(* CODESYS project Industy_RECOVERED_2026-05-19T08-51-21.project

Project tree, tasks and I/O mapping:
  Device : CODESYS Control Win V3 x64, CODESYS, version 3.5.22.10
    application Application
      libraries: Standard, 3.5.22.0 (System)
      task MainTask (cyclic, interval t#20ms, priority 1) calls PLC_PRG
      DUTs (Data Types)/
        data type ST_AreaStatus
      program PLC_PRG [ST]
      Processes/
        program POU_07_Packaging [ST]
        program POU_03_Dryer [ST]
        program POU_04_Shelling [ST]
        program POU_01_Receiving [ST]
        program POU_02_Husking [ST]
        program POU_06_Treating [ST]
        program POU_05_Conditioning [ST]
      Blocks/
        function block POU_Vibration_Sensor [ST]
        function block POU_Flow_Sensor [ST]
        function block POU_Motor [ST]
      Symbols
*)

// Device/Application/DUTs (Data Types)/ST_AreaStatus
TYPE ST_AreaStatus :
STRUCT
	Running : BOOL;
	Stopped : BOOL;
	Failure : BOOL;
	Counters : DINT;
END_STRUCT
END_TYPE

// Device/Application/PLC_PRG
PROGRAM PLC_PRG
VAR

END_VAR

POU_01_Receiving();
POU_02_Husking();
POU_03_Dryer();
POU_04_Shelling();
POU_05_Conditioning();
POU_06_Treating();
POU_07_Packaging();

END_PROGRAM

// Device/Application/Processes/POU_01_Receiving
PROGRAM POU_01_Receiving
VAR
	CNV_001 : POU_Motor();
	
	Process_State : DINT;
	H_Start_Process : BOOL;
	
	Weight_Load : REAL;
	Truck_Counter : DINT;
	
	Timer_Truck_Discharge : TON;
	
END_VAR

CNV_001();

CASE Process_State OF
	0: //Initial State - Stopped
		CNV_001.I_Auto_Start := FALSE;
		IF H_Start_Process THEN
			Process_State := 1;
		END_IF
		H_Start_Process := FALSE;
	
	1: //Weighting Truck
		IF Truck_Counter MOD 2 = 0 THEN
			Weight_Load := Weight_Load + 2568;
		ELSE
			Weight_Load := Weight_Load - 1432;
		END_IF
		Truck_Counter := Truck_Counter + 1;
		Process_State := 2;
		
	2: //Start Unloading Truck
		Timer_Truck_Discharge(IN := TRUE, PT := T#2M);
		CNV_001.I_Auto_Start := TRUE;
		IF Timer_Truck_Discharge.Q THEN //When Finished receiving
			CNV_001.I_Auto_Start := FALSE;
			Timer_Truck_Discharge.IN := FALSE;
			Process_State := 0;
		END_IF		
		
	ELSE //Error
		Process_State := -1;
END_CASE

END_PROGRAM

// Device/Application/Blocks/POU_Motor
FUNCTION_BLOCK PUBLIC POU_Motor
VAR_INPUT
	I_Auto_Start : BOOL;
END_VAR
VAR_OUTPUT
	O_Start_Motor : BOOL;
END_VAR
VAR
	
END_VAR

IF I_Auto_Start THEN
	O_Start_Motor := TRUE;
ELSE
	O_Start_Motor := FALSE;
END_IF

END_FUNCTION_BLOCK

// Device/Application/Processes/POU_02_Husking
PROGRAM POU_02_Husking

VAR
	Process_Status : DINT;
	Receiving_Status : DINT;
	CNV_002 : POU_Motor;
	HUS_001 : POU_Motor;
	Bins_Counter : DINT;
	
	Timer_End_of_Line : TON;

END_VAR

Receiving_Status := POU_01_Receiving.Process_State;

CASE Process_Status OF
	0: //Initial State - Stopped
		HUS_001.I_Auto_Start := FALSE;
		CNV_002.I_Auto_Start := FALSE;
		IF Receiving_Status = 1 THEN
			Process_Status := 1;
		END_IF

	1: //Starting Motors to husk 
		HUS_001.I_Auto_Start := TRUE;
		CNV_002.I_Auto_Start := TRUE;
		IF Receiving_Status = 2 THEN
			Process_Status := 2;
		END_IF
		
	2: //Husking Corn
		IF POU_01_Receiving.Timer_Truck_Discharge.Q THEN
			Timer_End_of_Line(IN := TRUE, PT := T#1M);
			IF Timer_End_of_Line.Q THEN
				HUS_001.I_Auto_Start := FALSE;
				CNV_002.I_Auto_Start := FALSE;
				Process_Status := 3;
			END_IF
		END_IF
		
	3: //Bin Dryer Full
		Bins_Counter := Bins_Counter + 1;
		Timer_End_of_Line.IN := FALSE;
		Process_Status := 0;
		
	ELSE //Error
		Process_Status := -1;		
END_CASE

END_PROGRAM

// Device/Application/Processes/POU_03_Dryer
PROGRAM POU_03_Dryer
VAR
	Husking_Status : DINT;
	Process_Status : DINT;
	Dryed_Bins : DINT;
	
	BLR_001 : POU_Motor;
	CNV_003 : POU_Motor;
	
	Air_Temp : REAL;
	Grain_Humidity : REAL;	
	
	Timer_End_of_Line : TON;
	Timer_Humi_Decreaser : TP;
	
	
END_VAR

Husking_Status := POU_02_Husking.Process_Status;

CASE Process_Status OF
	0: //Initial_Case - Stopped
		BLR_001.I_Auto_Start := FALSE;
		CNV_003.I_Auto_Start := FALSE;
		IF Husking_Status = 3 THEN
			Process_Status := 1;
		END_IF
		
	1: //Starting Dryer
		BLR_001.I_Auto_Start := TRUE;
		Grain_Humidity := 35.0;
		Air_Temp := 45.0;
		Process_Status := 2;
	2: //Drying Corn
		Timer_Humi_Decreaser(IN := NOT Timer_Humi_Decreaser.Q, PT := T#1M);
		WHILE Process_Status = 2 DO
			IF Grain_Humidity <= 13.0 AND Air_Temp = 45 THEN
				Process_Status := 3;
			ELSE
				IF Timer_Humi_Decreaser.Q THEN
					Grain_Humidity := Grain_Humidity - 0.35;					
				END_IF
			END_IF						
		END_WHILE
	
	3: // Corn Dry
		BLR_001.I_Auto_Start := FALSE;
		CNV_003.I_Auto_Start := TRUE;
		Timer_End_of_Line(IN := TRUE, PT := T#1M);
		IF Timer_End_of_Line.Q THEN
			CNV_003.I_Auto_Start := FALSE;
			Process_Status := 4;
		END_IF
		
	4: //Bin Empty
		Dryed_Bins := Dryed_Bins + 1;
		Timer_End_of_Line.IN := FALSE;
		Process_Status := 0;
		
	ELSE //Error
		Process_Status := -1;
END_CASE

END_PROGRAM

// Device/Application/Processes/POU_04_Shelling
PROGRAM POU_04_Shelling
VAR
	Dryer_Status : DINT;
	Process_Status : DINT;
	
	Sheller_RPM : REAL;
	Grain_Flow : REAL;
	
	SHL_001 : POU_Motor;
	CNV_004 : POU_Motor;
	
	Timer_Acc_Sheller : TP;
	Timer_End_of_Line : TON;
	
	Flow_Sensor : POU_Flow_Sensor;
	
END_VAR

Dryer_Status := POU_03_Dryer.Process_Status;
Flow_Sensor(Line_Status := Process_Status, Line_Nominal_Flow := 40.0);
SHL_001();
CNV_004();


CASE Process_Status OF
	0: //Initial Status - Stopped
		SHL_001.I_Auto_Start := FALSE;
		CNV_004.I_Auto_Start := FALSE;
		IF Dryer_Status = 3 THEN
			Process_Status := 1;
		END_IF
		
	1: //Start Sheller Motors
		CNV_004.I_Auto_Start := TRUE;
		SHL_001.I_Auto_Start := TRUE;
		Timer_Acc_Sheller(IN := NOT Timer_Acc_Sheller.Q, PT := T#1S);
		WHILE Process_Status = 1 DO
			IF Sheller_RPM = 40 THEN
				Process_Status := 2;
			ELSE
				IF Timer_Acc_Sheller.Q THEN
					Sheller_RPM := Sheller_RPM + 0.5;
				END_IF
			END_IF
		END_WHILE	
		
	2: //Start Shelling
		Grain_Flow := Flow_Sensor.Flow;
		Timer_End_of_Line(IN := TRUE, PT := T#1M);
		IF Timer_End_of_Line.Q THEN
			Process_Status := 3;
		END_IF
		
	3: //Finished Shelling
		SHL_001.I_Auto_Start := FALSE;
		CNV_004.I_Auto_Start := FALSE;
		Timer_Acc_Sheller(IN := NOT Timer_Acc_Sheller.Q, PT := T#1S);
		WHILE Process_Status = 3 DO
			IF Sheller_RPM <= 0 THEN
				Sheller_RPM := 0.0;
				Process_Status := 0;
			ELSE
				IF Timer_Acc_Sheller.Q THEN
					Sheller_RPM := Sheller_RPM - 2.3;
				END_IF
			END_IF
		END_WHILE
	ELSE //Error
		Process_Status := -1;
END_CASE

END_PROGRAM

// Device/Application/Blocks/POU_Flow_Sensor
FUNCTION_BLOCK POU_Flow_Sensor
VAR_INPUT
	Line_Status : DINT;
	Line_Nominal_Flow : REAL;
END_VAR
VAR_OUTPUT
	Flow : REAL;
END_VAR
VAR
	Signal_Noise : DINT;
END_VAR

IF NOT Line_Status <= 0 OR Line_Status >= 3 THEN
	Signal_Noise := Signal_Noise + 1;
	IF Signal_Noise > 10 THEN
		Signal_Noise := -10;
	END_IF
	Flow := Line_Nominal_Flow + (INT_TO_REAL(Signal_Noise)*0.15);
ELSE
	IF Flow > 0.0 THEN
		Flow := Flow - 2.5;
	ELSE
		Flow := 0;
	END_IF
END_IF

END_FUNCTION_BLOCK

// Device/Application/Processes/POU_05_Conditioning
PROGRAM POU_05_Conditioning
VAR
	Shelling_Process : DINT;
	Process_Status: DINT;

	CND_001 : POU_Motor;
	CND_002 : POU_Motor;
	CNV_005 : POU_Motor;
	
	Vibration_CND_001 : REAL;
	Vibration_CND_002 : REAL;
	
	Vibration_Sensor_CND_001 : POU_Vibration_Sensor;
	Vibration_Sensor_CND_002 : POU_Vibration_Sensor;
	
END_VAR

CND_001();
CND_002();
CNV_005();

Vibration_Sensor_CND_001(Motor_Started := CND_001.O_Start_Motor,Motor_Nominal_Vibration := 60);
Vibration_Sensor_CND_002(Motor_Started := CND_002.O_Start_Motor,Motor_Nominal_Vibration := 60);
Vibration_CND_001 := Vibration_Sensor_CND_001.Vibration;
Vibration_CND_002 := Vibration_Sensor_CND_001.Vibration;

Shelling_Process := POU_04_Shelling.Process_Status;

CASE Process_Status OF
	0: //Initial Status - Stopped
		CND_001.I_Auto_Start := FALSE;
		CND_002.I_Auto_Start := FALSE;
		CNV_005.I_Auto_Start := FALSE;
		IF Shelling_Process = 1 THEN
			Process_Status := 1;
		END_IF
		
	1: //Starting Motors
		CND_001.I_Auto_Start := TRUE;
		CND_002.I_Auto_Start := TRUE;
		CNV_005.I_Auto_Start := TRUE;
		Process_Status := 2;
		
	2: //Conditioning
		
		
		
		
END_CASE

END_PROGRAM

// Device/Application/Blocks/POU_Vibration_Sensor
FUNCTION_BLOCK POU_Vibration_Sensor
VAR_INPUT
	Motor_Started : BOOL;
	Motor_Nominal_Vibration : REAL;
END_VAR
VAR_OUTPUT
	Vibration : REAL;
END_VAR
VAR
	Signal_Noise : DINT;
END_VAR

IF NOT Motor_Started = TRUE THEN
	Signal_Noise := Signal_Noise + 1;
	IF Signal_Noise > 5 THEN
		Signal_Noise := -5;
	END_IF
	Vibration := Motor_Nominal_Vibration + (INT_TO_REAL(Signal_Noise)*0.2);
ELSE
	IF Vibration > 0.0 THEN
		Vibration := Vibration - 3.25;
	ELSE
		Vibration := 0;
	END_IF
END_IF

END_FUNCTION_BLOCK

// Device/Application/Processes/POU_06_Treating
PROGRAM POU_06_Treating
VAR
END_VAR

END_PROGRAM

// Device/Application/Processes/POU_07_Packaging
PROGRAM POU_07_Packaging
VAR
END_VAR

END_PROGRAM
